// TIA Portal V15 export
// export: Created 2018-06-04T11:32:33.0897578Z, ExportSetting WithDefaults, WithReadOnly, DisplayName Totally Integrated Automation Portal, DisplayVersion V15, DisplayName STEP 7 Professional, DisplayVersion V15, DisplayName WinCC Professional, DisplayVersion V15, DisplayName TIA Portal Openness, DisplayVersion V15
DATA_BLOCK "EM_Index"   // DB2
{ S7_Optimized_Access := 'FALSE' }
VERSION : 0.1
// stored: AutoNumber true, CodeModifiedDate 2018-06-04T11:31:36.2595073Z, CompileDate 2018-06-04T11:31:36.8205394Z, CreationDate 2018-06-04T11:30:27.8755959Z, InterfaceModifiedDate 2018-06-04T11:31:33.0593242Z, IsConsistent true, IsKnowHowProtected false, IsOnlyStoredInLoadMemory false, IsPLCDB false, IsWriteProtectedInAS false, ModifiedDate 2018-06-04T11:31:36.2595073Z, ParameterModified 2018-06-04T11:31:33.0593242Z, StructureModified 2018-06-04T11:31:33.0593242Z
   VAR RETAIN
      DB_Numbers : Array[0..990] of Int;   // DB numbers of the EMs
   END_VAR
BEGIN
END_DATA_BLOCK
